// TwinCAT 3 PLC project PLC_ST01
// ProgramVersion: 3.1.4024.0
// libraries:
//   Base Objects Library, * (JABIL RAC LATAM)
//   Tc2_MC2, * (Beckhoff Automation GmbH)
//   Tc2_Standard, * (Beckhoff Automation GmbH)
//   Tc2_System, * (Beckhoff Automation GmbH)
//   Tc3_Module, * (Beckhoff Automation GmbH)
// project tree:
//   / PlcST01Task.TcTTO
//   POUs/00-MainPRG/ MAIN_ST01.TcPOU
//   POUs/01-FunctionBlocks/MaterialAssembly/ FB_ControllerAsm.TcPOU, FB_EndcapAsm.TcPOU
//   POUs/01-FunctionBlocks/MaterialSupply/ FB_BatterySupply.TcPOU, FB_ControllerSupply.TcPOU, FB_LoadStation.TcPOU
// real-time tasks:
//   TASK PlcST01Task: cycle T#10ms, priority 20, ADS port 350
//   TASK PlcST02Task: cycle T#10ms, priority 21, ADS port 351
//   TASK PlcST03Task: cycle T#10ms, priority 22, ADS port 352
// motion (NC):
//   TASK NC-Task 1 SAF: cycle T#2ms, priority 4, ADS port 501
//   TASK NC-Task 1 SVB: cycle T#10ms, priority 8, ADS port 511
//   AXIS Axis 1 (id 1)
//     OtherSettings: AllowMotionCmdToSlave=true
//     encoder EncType=19
//       EncPara: MaxCount=#xffffffff
//     drive DrvType=16
//       DrvPara: MaxCount=#xffffffff, DriveControlDWord=#x00000100
//         Analog: TorqueSetpointScale=10, ScaleFactorActTorque=0.1
//         TimeComp: TaskDelayCycles=1
//     controller CtrType=1
//       CtrPara: PriorControlFactor=1
//         Observer: BandWidth=20
//   AXIS Axis 2 (id 2)
//     OtherSettings: AllowMotionCmdToSlave=true
//     encoder EncType=19
//       EncPara: MaxCount=#xffffffff
//     drive DrvType=16
//       DrvPara: MaxCount=#xffffffff, DriveControlDWord=#x00000100
//         Analog: TorqueSetpointScale=10, ScaleFactorActTorque=0.1
//         TimeComp: TaskDelayCycles=1
//     controller CtrType=1
//       CtrPara: PriorControlFactor=1
//         Observer: BandWidth=20
//   AXIS Axis 3 (id 3)
//     OtherSettings: AllowMotionCmdToSlave=true
//     encoder EncType=19
//       EncPara: MaxCount=#xffffffff
//     drive DrvType=16
//       DrvPara: MaxCount=#xffffffff, DriveControlDWord=#x00000100
//         Analog: TorqueSetpointScale=10, ScaleFactorActTorque=0.1
//         TimeComp: TaskDelayCycles=1
//     controller CtrType=1
//       CtrPara: PriorControlFactor=1
//         Observer: BandWidth=20
// I/O:
//   DEVICE Device 1 (EtherCAT), AmsNetId 192.168.0.6.4.1
//     Term 1 (EK1100) [EK1100 EtherCAT Coupler (2A E-Bus)]
//       Term 2 (EL6910) [EL6910, TwinSAFE PLC]
//       Term 3 (EL1904) [EL1904, 4 Ch. Safety Input 24V, TwinSAFE]
//         modules: Module 1 (FSOES)
//       Term 4 (EL1904) [EL1904, 4 Ch. Safety Input 24V, TwinSAFE]
//         modules: Module 1 (FSOES)
//       Term 5 (EL1904) [EL1904, 4 Ch. Safety Input 24V, TwinSAFE]
//         modules: Module 1 (FSOES)
//       Term 6 (EL1904) [EL1904, 4 Ch. Safety Input 24V, TwinSAFE]
//         modules: Module 1 (FSOES)
//       Term 7 (EL1904) [EL1904, 4 Ch. Safety Input 24V, TwinSAFE]
//         modules: Module 1 (FSOES)
//       Term 8 (EL1904) [EL1904, 4 Ch. Safety Input 24V, TwinSAFE]
//         modules: Module 1 (FSOES)
//       Term 9 (EL1904) [EL1904, 4 Ch. Safety Input 24V, TwinSAFE]
//         modules: Module 1 (FSOES)
//       Term 10 (EL1904) [EL1904, 4 Ch. Safety Input 24V, TwinSAFE]
//         modules: Module 1 (FSOES)
//       Term 11 (EL9410) [EL9410 E-Bus Power Supplier  (Diagnostics)]
//       Term 12 (EL2904) [EL2904, 4 Ch. Safety Output 24V, 0.5A, TwinSAFE]
//         modules: Module 1 (FSOES), Module 2 (DO)
//       Term 13 (EL2904) [EL2904, 4 Ch. Safety Output 24V, 0.5A, TwinSAFE]
//         modules: Module 1 (FSOES), Module 2 (DO)
//       Term 14 (EL2904) [EL2904, 4 Ch. Safety Output 24V, 0.5A, TwinSAFE]
//         modules: Module 1 (FSOES), Module 2 (DO)
//       Term 15 (EL2904) [EL2904, 4 Ch. Safety Output 24V, 0.5A, TwinSAFE]
//         modules: Module 1 (FSOES), Module 2 (DO)
//       Term 16 (EL1809) [EL1809 16Ch. Dig. Input 24V, 3ms]
//       Term 17 (EL1809) [EL1809 16Ch. Dig. Input 24V, 3ms]
//       Term 18 (EL1809) [EL1809 16Ch. Dig. Input 24V, 3ms]
//       Term 19 (EL1809) [EL1809 16Ch. Dig. Input 24V, 3ms]
//       Term 20 (EL1809) [EL1809 16Ch. Dig. Input 24V, 3ms]
//       Term 21 (EL1809) [EL1809 16Ch. Dig. Input 24V, 3ms]
//       Term 22 (EL1809) [EL1809 16Ch. Dig. Input 24V, 3ms]
//       Term 23 (EL9410) [EL9410 E-Bus Power Supplier  (Diagnostics)]
//       Term 24 (EL1809) [EL1809 16Ch. Dig. Input 24V, 3ms]
//       Term 25 (EL1809) [EL1809 16Ch. Dig. Input 24V, 3ms]
//       Term 26 (EL1809) [EL1809 16Ch. Dig. Input 24V, 3ms]
//       Term 27 (EL2809) [EL2809 16Ch. Dig. Output 24V, 0.5A]
//       Term 28 (EL2809) [EL2809 16Ch. Dig. Output 24V, 0.5A]
//       Term 29 (EL2809) [EL2809 16Ch. Dig. Output 24V, 0.5A]
//       Term 30 (EL2809) [EL2809 16Ch. Dig. Output 24V, 0.5A]
//       Term 31 (EL2809) [EL2809 16Ch. Dig. Output 24V, 0.5A]
//       Term 32 (EL2809) [EL2809 16Ch. Dig. Output 24V, 0.5A]
//       Term 33 (EL2809) [EL2809 16Ch. Dig. Output 24V, 0.5A]
//       Term 34 (EL2809) [EL2809 16Ch. Dig. Output 24V, 0.5A]
//       Term 35 (EL3062) [EL3062 2Ch. Ana. Input 0-10V]
//       Term 36 (EL6652) [EL6652 EtherNet/IP Scanner (Master)]
//       Term 40 (EL9011) [EL9011 End Terminal]
//     Drive 37 (MDDLT55BF) [MDDLT55BF]
//     Drive 38 (MADLT05BF) [MADLT05BF]
//     Drive 39 (MADLT05BF) [MADLT05BF]
//   DEVICE Device 1 (ECAT EIP Scanner (EL6652)), AmsNetId 192.168.0.6.2.1
//     Robot01_Controller // <INFO> 192.168.0.21, ABB Adapter (ProdCode: 1, Rev: 2.50, Mac: 74:fe:48:88:fe:f3) </INFO> <EDS> C:\TwinCAT\3.1\Config\Io\EtherNetIP\enip.eds </EDS>
//     Robot02_Battery // <INFO> 192.168.0.22, ABB Adapter (ProdCode: 1, Rev: 2.50, Mac: 74:fe:48:87:d9:ae) </INFO> <EDS> C:\TwinCAT\3.1\Config\Io\EtherNetIP\enip.eds </EDS>
//     Robot03_1-2 // <INFO> 192.168.0.23, ABB Adapter (ProdCode: 1, Rev: 2.50, Mac: 74:fe:48:88:fe:f0) </INFO> <EDS> C:\TwinCAT\3.1\Config\Io\EtherNetIP\enip.eds </EDS>
//     Robot04_2-3 // <INFO> 192.168.0.24, ABB Adapter (ProdCode: 1, Rev: 2.50, Mac: 74:fe:48:88:0a:25) </INFO> <EDS> C:\TwinCAT\3.1\Config\Io\EtherNetIP\enip.eds </EDS>
//     NX1P2_ControllerTFPLC // <INFO> 192.168.0.10, NX1P2 (ProdCode: 1675, Rev: 2.09, Mac: 3c:f7:d1:1e:14:dc) </INFO> <EDS> C:\TwinCAT\3.1\Config\Io\EtherNetIP\ </EDS>
//     NX1P2_BatteryTrayFeederPLC // <INFO> 192.168.0.13, NX1P2 (ProdCode: 1675, Rev: 2.09, Mac: 3c:f7:d1:16:20:93) </INFO> <EDS> C:\TwinCAT\3.1\Config\Io\EtherNetIP\ </EDS>
// variable links:
//   NC-Task 1 SAF/Axes/Axis 1 <-> Device 1 (EtherCAT)/Drive 37 (MDDLT55BF)
//     Drive/Inputs/In/nDataIn1 <-> Transmit PDO mapping 1/Following error actual value
//     Drive/Inputs/In/nState1 <-> Transmit PDO mapping 1/Statusword
//     Drive/Inputs/In/nState2 <-> Transmit PDO mapping 1/Statusword @bit 8
//     Drive/Inputs/In/nState4 @bit 1 <-> WcState/InputToggle
//     Drive/Inputs/In/nState4 <-> WcState/WcState
//     Drive/Inputs/In/nState5 <-> Transmit PDO mapping 1/Modes of operation display
//     Drive/Outputs/Out/nCtrl1 <-> Receive PDO mapping 1/Controlword
//     Drive/Outputs/Out/nCtrl2 <-> Receive PDO mapping 1/Controlword @bit 8
//     Drive/Outputs/Out/nCtrl5 <-> Receive PDO mapping 1/Modes of operation
//     Drive/Outputs/Out/nDataOut1 <-> Receive PDO mapping 1/Target position
//     Enc/Inputs/In/nDataIn1 <-> Transmit PDO mapping 1/Position actual value
//     Enc/Inputs/In/nDataIn3 <-> Transmit PDO mapping 1/Touch probe pos1 pos value
//     Enc/Inputs/In/nState4 @bit 1 <-> WcState/InputToggle
//     Enc/Inputs/In/nState4 <-> WcState/WcState
//     Enc/Inputs/In/nState5 <-> Transmit PDO mapping 1/Touch probe status
//     Enc/Inputs/In/nState6 <-> Transmit PDO mapping 1/Touch probe status @bit 8
//     Enc/Outputs/Out/nCtrl5 <-> Receive PDO mapping 1/Touch probe function
//     Enc/Outputs/Out/nCtrl6 <-> Receive PDO mapping 1/Touch probe function @bit 8
//   NC-Task 1 SAF/Axes/Axis 2 <-> Device 1 (EtherCAT)/Drive 38 (MADLT05BF)
//     Drive/Inputs/In/nDataIn1 <-> Transmit PDO mapping 1/Following error actual value
//     Drive/Inputs/In/nState1 <-> Transmit PDO mapping 1/Statusword
//     Drive/Inputs/In/nState2 <-> Transmit PDO mapping 1/Statusword @bit 8
//     Drive/Inputs/In/nState4 @bit 1 <-> WcState/InputToggle
//     Drive/Inputs/In/nState4 <-> WcState/WcState
//     Drive/Inputs/In/nState5 <-> Transmit PDO mapping 1/Modes of operation display
//     Drive/Outputs/Out/nCtrl1 <-> Receive PDO mapping 1/Controlword
//     Drive/Outputs/Out/nCtrl2 <-> Receive PDO mapping 1/Controlword @bit 8
//     Drive/Outputs/Out/nCtrl5 <-> Receive PDO mapping 1/Modes of operation
//     Drive/Outputs/Out/nDataOut1 <-> Receive PDO mapping 1/Target position
//     Enc/Inputs/In/nDataIn1 <-> Transmit PDO mapping 1/Position actual value
//     Enc/Inputs/In/nDataIn3 <-> Transmit PDO mapping 1/Touch probe pos1 pos value
//     Enc/Inputs/In/nState4 @bit 1 <-> WcState/InputToggle
//     Enc/Inputs/In/nState4 <-> WcState/WcState
//     Enc/Inputs/In/nState5 <-> Transmit PDO mapping 1/Touch probe status
//     Enc/Inputs/In/nState6 <-> Transmit PDO mapping 1/Touch probe status @bit 8
//     Enc/Outputs/Out/nCtrl5 <-> Receive PDO mapping 1/Touch probe function
//     Enc/Outputs/Out/nCtrl6 <-> Receive PDO mapping 1/Touch probe function @bit 8
//   NC-Task 1 SAF/Axes/Axis 3 <-> Device 1 (EtherCAT)/Drive 39 (MADLT05BF)
//     Drive/Inputs/In/nDataIn1 <-> Transmit PDO mapping 1/Following error actual value
//     Drive/Inputs/In/nState1 <-> Transmit PDO mapping 1/Statusword
//     Drive/Inputs/In/nState2 <-> Transmit PDO mapping 1/Statusword @bit 8
//     Drive/Inputs/In/nState4 @bit 1 <-> WcState/InputToggle
//     Drive/Inputs/In/nState4 <-> WcState/WcState
//     Drive/Inputs/In/nState5 <-> Transmit PDO mapping 1/Modes of operation display
//     Drive/Outputs/Out/nCtrl1 <-> Receive PDO mapping 1/Controlword
//     Drive/Outputs/Out/nCtrl2 <-> Receive PDO mapping 1/Controlword @bit 8
//     Drive/Outputs/Out/nCtrl5 <-> Receive PDO mapping 1/Modes of operation
//     Drive/Outputs/Out/nDataOut1 <-> Receive PDO mapping 1/Target position
//     Enc/Inputs/In/nDataIn1 <-> Transmit PDO mapping 1/Position actual value
//     Enc/Inputs/In/nDataIn3 <-> Transmit PDO mapping 1/Touch probe pos1 pos value
//     Enc/Inputs/In/nState4 @bit 1 <-> WcState/InputToggle
//     Enc/Inputs/In/nState4 <-> WcState/WcState
//     Enc/Inputs/In/nState5 <-> Transmit PDO mapping 1/Touch probe status
//     Enc/Inputs/In/nState6 <-> Transmit PDO mapping 1/Touch probe status @bit 8
//     Enc/Outputs/Out/nCtrl5 <-> Receive PDO mapping 1/Touch probe function
//     Enc/Outputs/Out/nCtrl6 <-> Receive PDO mapping 1/Touch probe function @bit 8
//   PLC_ST01/PLC_ST01 Instance <-> Device 1 (ECAT EIP Scanner (EL6652))/Robot02_Battery
//     PlcST01Task Inputs/MAIN_ST01.fbBatterySupply.fbRobot.RobotIO.eipInputs <-> Connection 2 (Input/Output)/Inputs/inputRaw

CONFIGURATION PLC_ST01
    RESOURCE PLC ON TwinCAT3
        TASK PlcST01Task(INTERVAL := T#10ms, PRIORITY := 20);
        PROGRAM MAIN_ST01 WITH PlcST01Task : MAIN_ST01;
    END_RESOURCE
END_CONFIGURATION

// ---- POUs/00-MainPRG/MAIN_ST01.TcPOU
PROGRAM MAIN_ST01
VAR
	fbStation01							: RACBaseObjects.FB_Station;
	fbConveyor							: RACBaseObjects.FB_Conveyor;
	fbControllerSupply					: FB_ControllerSupply;
	fbBatterySupply						: FB_BatterySupply;
	fbEndcapAsm							: FB_EndcapAsm;
	fbControllerAsm						: FB_ControllerAsm;
	fbLoadStation						: FB_LoadStation;
	
	// Input from ST02
	ST02_initFinished					AT%I* : BOOL;
	ST02_mtrlReq						AT%I* : BOOL;
	
	// Estop declaration
	bEStopLoad							AT%I*	: BOOL;
	bEStopUserInterface					AT%I*	: BOOL;
	
	// Door no contact declaration
	
	// Interlock inputs declaration
	
END_VAR

	fbStation01(						bInitFinished:=fbControllerSupply.bInit_Finished AND fbBatterySupply.bInit_Finished AND fbConveyor.bInit_Finished,
										EmergencyStop:=bEStopLoad OR bEStopUserInterface,
										safetyReady:=TRUE,
										Interlock:=TRUE);

	fbConveyor(							sDeviceID:='',
										bStopExecution:=fbStation01.bStop,
										bAlarmReset:=fbStation01.bAlarmReset,
										diStationState:=fbStation01.diStationState,
										bInit_StartPermissive:=fbLoadStation.bInit_Finished AND fbEndcapAsm.bInit_Finished AND fbControllerAsm.bInit_Finished AND fbBatterySupply.bInit_Finished AND ST02_initFinished,
										bIn_SafeToMove:=FALSE,
										bIn_AllProcessComplete:=FALSE,
										lrDistance:=0,
										lrOffsetPos:=0,
										bIn_IsClamped:=FALSE,
										bIn_IsUnclamped:=FALSE);

	fbLoadStation(						sDeviceID:='',
										bStopExecution:=fbStation01.bStop,
										bAlarmReset:=fbStation01.bAlarmReset,
										diStationState:=fbStation01.diStationState,
										bInit_StartPermissive := TRUE,
										bDisableScan := TRUE,
										bIn_MovePermisive := FALSE,
										bIn_CvyStepDone := FALSE);

	fbEndcapAsm(						sDeviceID:='',
										bStopExecution:=fbStation01.bStop,
										bAlarmReset:=fbStation01.bAlarmReset,
										diStationState:=fbStation01.diStationState,
										bInit_StartPermissive:=TRUE,
										bSafetyBoxPlace_permissive :=TRUE);
	
										
	fbControllerSupply(					sDeviceID:='',
										bStopExecution:=fbStation01.bStop,
										bAlarmReset:=fbStation01.bAlarmReset,
										diStationState:=fbStation01.diStationState,
										bInit_StartPermissive:=TRUE,
										bSafetyBoxPlace_permissive:=FALSE,
										bPlace_MaterialRequest:=FALSE);
										
	fbControllerAsm(					sDeviceID:='',
										bStopExecution:=fbStation01.bStop,
										bAlarmReset:=fbStation01.bAlarmReset,
										diStationState:=fbStation01.diStationState,
										bInit_StartPermissive:=TRUE,
										sSerialReceived:=fbControllerSupply.sPieceSN,	
										bIn_RailReady:=fbConveyor.bOut_MoveDone);
										
	fbBatterySupply(					sDeviceID:='',
										bStopExecution:=fbStation01.bStop,
										bAlarmReset:=fbStation01.bAlarmReset,
										diStationState:=fbStation01.diStationState,
										bInit_StartPermissive:=TRUE,
										bSafetyBoxPlace_permissive := FALSE,
										bPlace_MaterialRequest := TRUE);

END_PROGRAM

// ---- POUs/01-FunctionBlocks/MaterialSupply/FB_ControllerSupply.TcPOU
FUNCTION_BLOCK FB_ControllerSupply EXTENDS RACBaseObjects.FB_Machine
VAR_INPUT
	bSafetyBoxPlace_Permissive			: BOOL;
	bPlace_MaterialRequest				: BOOL;
END_VAR
VAR_OUTPUT
	bSafetyBoxPlace_OutOfZone			: BOOL;
	sPieceSN							: STRING;
	bPlace_Done							: BOOL;
END_VAR
VAR
	fbTrayFeeder						: RACBaseObjects.FB_TrayFeeder;
	fbRobot								: RACBaseObjects.FB_Robot;
	fbScanner							: RACBaseObjects.FB_Scanner;
	
	// Reject on belt in tray feeder safery box permissive
	bSafetyBoxReject_permissive			AT%I*	: BOOL;
	// Reject on belt in tray feeder material request
	bReject_MaterialRequest				AT%I*	: BOOL;
	// Reject on belt in tray feeder out of safery box
	bSafetyBoxReject_OutOfZone			AT%Q*	: BOOL;
	// Reject on belt in tray feeder reject done
	bReject_Done						AT%Q*	: BOOL;
	
	// Auto procees is scanning
	bScann								: BOOL;
	
	// OK esponse from Acuram MES consultimng
	bPieceIsGood						: BOOL;
	// NG esponse from Acuram MES consultimng
	bPieceIsNG							: BOOL;
	
	// Auxiliar bool array for reject places inputs
	bAvailableNests						: ARRAY[0..7] OF BOOL;
END_VAR

SUPER^.MachineMain();
//	Tray Feeder instance
	fbTrayFeeder(						sDeviceID:=	'01',
										bStopExecution:=bStopExecution,
										bAlarmReset:=bAlarmReset,
										diStationState:=diStationState,
										bInit_StartPermissive:=fbRobot.bInit_Finished,
										bSafetyBoxDeliver_permissive:=fbRobot.bSafetyBoxPick_OutOfZone,
										bChangeTrayRequest:=fbRobot.bPick_AllMaterialPicked);

//	Robot instance
	fbRobot(							sDeviceID:=	'01',
										bStopExecution:=bStopExecution,
										bAlarmReset:=bAlarmReset,
										diStationState:=diStationState,
										bInit_StartPermissive:=bInit_StartPermissive,
										bSafetyBoxPick_Permissive:=fbTrayFeeder.bSafetyBoxDeliver_isSafe,
										bSafetyBoxPlace_Permissive:=bSafetyBoxPlace_permissive,
										bSafetyBoxReject_Permissive:=bSafetyBoxReject_Permissive,
										bOKMaterialReadyToPick:=fbTrayFeeder.bMaterial_ReadyToPick,
										bNGMaterialReadyToPick:=FALSE,
										bPiceIsGood:=bPieceIsGood,
										bPiceIsNG:=bPieceIsNG,
										bPlace_MaterialRequest:=bPlace_MaterialRequest,
										bReject_MaterialRequest:=bAvailableNests,
										bSafetyBoxPlace_OutOfZone=>bSafetyBoxPlace_OutOfZone,
										bSafetyBoxReject_OutOfZone=>bSafetyBoxReject_OutOfZone,
										bPlace_Done=>bPlace_Done,
										bReject_Done=>bReject_Done);

//	Scanner insance
	fbScanner(							sDeviceID:=	'03',
										bStopExecution:=bStopExecution,
										bAlarmReset:=bAlarmReset,
										bIn_Trigger:=bScann,
										bDisable:=FALSE,
										iTotalRetries:=2,
										Timeout:=t#1s);

METHOD Alarm
sAlarm:= CONCAT(STR1:=fbTrayFeeder.sAlarm, STR2:=fbRobot.sAlarm);
sAlarm:= CONCAT(STR1:=sAlarm,STR2:=fbScanner.sAlarm);
END_METHOD

METHOD Auto
//	When finish reading save the code in a var
	IF (fbRobot.diActualSeqStep=EN_RobotMessaging.waitingPieceStatus) THEN
		bScann:=TRUE;
		IF (fbScanner.bCompleted) AND (sPieceSN<>fbScanner.sCode) THEN
			sPieceSN:=fbScanner.sCode;
		END_IF
	END_IF

//	For clearing code in var
	IF (fbRobot.diActualSeqStep<>EN_RobotMessaging.waitingPieceStatus) AND (fbRobot.diActualSeqStep<>EN_RobotMessaging.placing) AND (fbRobot.diActualSeqStep<>EN_RobotMessaging.placeFinished) THEN
		bPieceIsGood:=FALSE;
		bPieceIsNG:=FALSE;
		sPieceSN:='';
	END_IF
END_METHOD

METHOD Init
bInit_Finished:=fbTrayFeeder.bInit_Finished AND fbRobot.bInit_Finished AND fbScanner.bConnected;
END_METHOD

METHOD IO
//	For robot available places inputs
	bAvailableNests[0]					:= bReject_MaterialRequest;
	bAvailableNests[1]					:= FALSE;
	bAvailableNests[2]					:= FALSE;
	bAvailableNests[3]					:= FALSE;
	bAvailableNests[4]					:= FALSE;
	bAvailableNests[5]					:= FALSE;
	bAvailableNests[6]					:= FALSE;
	bAvailableNests[7]					:= FALSE;
END_METHOD

{warning 'Add method implementation '}
METHOD Manual
END_METHOD

{warning 'Add method implementation '}
METHOD Pause
END_METHOD

{warning 'Add method implementation '}
METHOD Stop
END_METHOD

END_FUNCTION_BLOCK

// ---- POUs/01-FunctionBlocks/MaterialSupply/FB_BatterySupply.TcPOU
FUNCTION_BLOCK FB_BatterySupply EXTENDS RACBaseObjects.FB_Machine
VAR_INPUT
	bSafetyBoxPlace_permissive			: BOOL;
	
	bPlace_MaterialRequest				: BOOL;
END_VAR
VAR_OUTPUT
	bSafetyBoxPlace_OutOfZone			: BOOL;
	
	sPieceSN							: STRING;
	sPieceOnGantrySN					: STRING;
	sPieceOnSliderSN					: STRING;
	
	bPlace_Done							: BOOL;
END_VAR
VAR
	fbTrayFeeder						: RACBaseObjects.FB_TrayFeeder;
	fbRobot								: RACBaseObjects.FB_Robot;
	fbScanner							: RACBaseObjects.FB_Scanner;
	
	// Auto procees is scanning
	bScann								: BOOL;
	
	// Auxiliar bool array for reject places inputs
	bAvailableNests						: ARRAY[0..7] OF BOOL;
END_VAR

SUPER^.MachineMain();
//	Tray Feeder instance
	fbTrayFeeder(						sDeviceID:=	'',
										bStopExecution:=bStopExecution,
										bAlarmReset:=bAlarmReset,
										diStationState:=diStationState,
										bInit_StartPermissive:=fbRobot.bInit_Finished,
										bSafetyBoxDeliver_permissive:=fbRobot.bSafetyBoxPick_OutOfZone,
										bChangeTrayRequest:=fbRobot.bPick_AllMaterialPicked);

//	Robot instance
//	fbRobot(							sDeviceID:=	'',
//										bStopExecution:=bStopExecution,
//										bAlarmReset:=bAlarmReset,
//										diStationState:=diStationState,
//										bInit_StartPermissive:=bInit_StartPermissive,
//										bSafetyBoxPick_Permissive:=fbTrayFeeder.bSafetyBoxDeliver_isSafe,
//										bSafetyBoxPlace_Permissive:=bSafetyBoxPlace_permissive,
//										bSafetyBoxReject_Permissive:=FALSE,
//										bOKMaterialReadyToPick:=fbTrayFeeder.bMaterial_ReadyToPick,
//										bNGMaterialReadyToPick:=FALSE,
//										bPiceIsGood:=TRUE,
//										bPiceIsNG:=FALSE,
//										bPlace_MaterialRequest:=bPlace_MaterialRequest,
//										bReject_MaterialRequest:=bAvailableNests,
//										bSafetyBoxPlace_OutOfZone=>bSafetyBoxPlace_OutOfZone,
//										bPlace_Done=>bPlace_Done);

//	Scanner insance
	fbScanner(							sDeviceID:=	'',
										bStopExecution:=bStopExecution,
										bAlarmReset:=bAlarmReset,
										bIn_Trigger:=bScann,
										bDisable:=FALSE,
										iTotalRetries:=2,
										Timeout:=t#1s);

METHOD Alarm
sAlarm:= CONCAT(STR1:=fbTrayFeeder.sAlarm, STR2:=fbRobot.sAlarm);
sAlarm:= CONCAT(STR1:=sAlarm,STR2:=fbScanner.sAlarm);
END_METHOD

METHOD Auto
VAR
END_VAR
//	When slider is not taking piece, reaching delivery position or delivering unit, clear piece on slider code var
	IF (fbTrayFeeder.diActualSeqStep<>1110) AND (fbTrayFeeder.diActualSeqStep<>1120) AND (fbTrayFeeder.diActualSeqStep<>1130) THEN
		sPieceSN:='';
	END_IF

//	When finish reading save the code in a var
	IF fbTrayFeeder.diActualSeqStep=1110 THEN
		bScann:=TRUE;
		IF (fbScanner.bCompleted) AND (sPieceSN<>fbScanner.sCode) THEN
			sPieceSN:=fbScanner.sCode;
		END_IF
	END_IF

//	When gantry takes the battery translate last serial code readed
	IF (fbTrayFeeder.diActualSeqStep=1130) AND (sPieceOnGantrySN=sPieceSN) THEN
		sPieceOnGantrySN:=sPieceSN;
	END_IF

//	When gantry release the battery translate serial code to other var
	IF (fbTrayFeeder.diActualSeqStep=1150) AND (sPieceOnSliderSN<>sPieceOnGantrySN) THEN
		sPieceOnSliderSN:=sPieceOnGantrySN;
	END_IF
END_METHOD

METHOD Init
bInit_Finished:=fbTrayFeeder.bInit_Finished AND fbRobot.bInit_Finished AND fbScanner.bConnected;
END_METHOD

METHOD IO
//	For robot available places inputs
	bAvailableNests[0]					:= FALSE;
	bAvailableNests[1]					:= FALSE;
	bAvailableNests[2]					:= FALSE;
	bAvailableNests[3]					:= FALSE;
	bAvailableNests[4]					:= FALSE;
	bAvailableNests[5]					:= FALSE;
	bAvailableNests[6]					:= FALSE;
	bAvailableNests[7]					:= FALSE;
END_METHOD

{warning 'Add method implementation '}
METHOD Manual
END_METHOD

{warning 'Add method implementation '}
METHOD Pause
END_METHOD

{warning 'Add method implementation '}
METHOD Stop
END_METHOD

END_FUNCTION_BLOCK

// ---- POUs/01-FunctionBlocks/MaterialAssembly/FB_EndcapAsm.TcPOU
FUNCTION_BLOCK INTERNAL FB_EndcapAsm EXTENDS RACBaseObjects.FB_Machine
VAR_INPUT
	bSafetyBoxPlace_permissive			: BOOL;
END_VAR
VAR_OUTPUT
	bOutEndcapAsm_Done 					: BOOL;
END_VAR
VAR
	bIsEndcapInFeedPosition		AT %I*		: BOOL;
	bIsEndcapInAssemblyPos		AT %I*		: BOOL;
	bFirstPositionSensor 		AT %I*		: BOOL;		
				
	//Is rail in position and clamped
	bRailReadyToAssembly					: BOOL;
	//Assembly side is ready to receive
	bAsmReadyToReceive						: BOOL;
	//Feed side with endcap ready
	bFeedReadyToSend						: BOOL;
	//The endcap is assembled on the rail
	bEndcapInRailDone						: BOOL;
	
	//Local process control
	bRemoveBottomSupport					: BOOL;
	bEndcapAssembled						: BOOL;
	bIsClampedOk							: BOOL;
	bIsReleased								: BOOL;
	bIsBottomClampRelease					: BOOL;								
	bEndcapPasses							: BOOL;		
	
	//Control steps for sub routines
	iStepAsm								: USINT;
	iStepFeed								: USINT;
	iStepRail								: USINT;
	
	//Timer to confirm endcap in position
	tmrPosition								: TON;
	tmrBowl									: TP;
	time_EC_DelayPosition					: TIME		:= T#500MS;
		
	//Devices
	
	//Bowl control structure, validate signals and control system1		
	bowlControl								: ST_BowlFeeder;	
	//Rail side for clamp support top cylinder
	Cyl_ClampRail_Top						: FB_Cylinder;
	//Rail side for clamp support bottom cylinder
	Cyl_ClampRail_Bot						: FB_Cylinder;		
	//Send endcap from bowl rail to assembly align
	Cyl_FeedEndcap							: FB_Cylinder;	
	//Push endcap for assembly with the rail 
	Cyl_PushEndcap							: FB_Cylinder;	
	//Endcap feeding guide during alignment process
	Cyl_SupportEndcap_Top					: FB_Cylinder;
	//Bottom alignment guide and pin button release 
	Cyl_SupportEndcap_Bot					: FB_Cylinder;

	bOut_ProcessComplete					: BOOL;
	bOut_ProcessOnFail						: BOOL;
	bOut_ReadyToReceive						: BOOL;
	bIn_UnitReady							: BOOL;
	bIn_UnitOnFail							: BOOL;
	
	//Manual operations
	bIn_Manual_ClampRail				: BOOL;
	bIn_Manual_UnclampRail				: BOOL;	
	bIn_ManualRun						: BOOL;		
	
	
END_VAR

SUPER^.MachineMain();

//Run FB and assign safety permisives


Cyl_ClampRail_Top();

Cyl_ClampRail_Bot();

//Set the permisive output directly from the cylinder sensors
bSafetyBoxPlace_Permissive := (Cyl_ClampRail_Top.bIsRetracted AND
							Cyl_ClampRail_Bot.bIsRetracted AND
							Cyl_PushEndcap.bIsRetracted);

METHOD Alarm
END_METHOD

METHOD Auto

VAR
	Seq_Endcap: INT;
END_VAR
//Call sub process
THIS^.Seq_EndcapFeed(bIsManual := TRUE);			//Feed endcap from bowl to assembly process
THIS^.Seq_EndcapAsm(bIsManual := TRUE);			//Endcap assembly process
THIS^.Seq_Auto_Rail();			//Clamp rail
THIS^.Seq_Auto_BowlFeeder();	//Bowl feeder control
END_METHOD

METHOD ClampRail : BOOL
//Top and bottom clamp
Cyl_ClampRail_Top.bExtendRequest:= TRUE;
Cyl_ClampRail_Bot.bExtendRequest:= TRUE;

ClampRail:=  Cyl_ClampRail_Top.bIsExtended AND Cyl_ClampRail_Bot.bIsExtended;
END_METHOD

METHOD fn_CancelCylinderMoves
VAR
	r_trig					: R_TRIG;
END_VAR
r_trig(CLK:= TRUE);
//Stop moves only once
IF r_trig.Q THEN
				
	Cyl_ClampRail_Bot.bExtendRequest:= FALSE;
	Cyl_ClampRail_Bot.bRetractRequest:= FALSE;
	
	Cyl_ClampRail_Top.bExtendRequest:= FALSE;
	Cyl_ClampRail_Top.bRetractRequest:= FALSE;
	
	Cyl_FeedEndcap.bExtendRequest:= FALSE;
	Cyl_FeedEndcap.bRetractRequest:= FALSE;
	
	Cyl_PushEndcap.bExtendRequest:= FALSE;
	Cyl_PushEndcap.bRetractRequest:= FALSE;
	
	Cyl_SupportEndcap_Bot.bExtendRequest:= FALSE;
	Cyl_SupportEndcap_Bot.bRetractRequest:= FALSE;
	
	Cyl_SupportEndcap_Top.bExtendRequest:= FALSE;
	Cyl_SupportEndcap_Top.bRetractRequest:= FALSE;
END_IF
END_METHOD

 METHOD Init 

//VAR_OUTPUT
//	bOutReadyToRobotPlace: BOOL;
//END_VAR
CASE diActualSeqStep OF
	//Initial
		
	0:						//Reset variables		
		bInit_Finished := FALSE;
	     bOutEndcapAsm_Done:= FALSE;		
		diActualSeqStep:= 10;	
		
	10:						//Retract rail support				
		//Retract controller guide support
		Cyl_SupportEndcap_Top.bRetractRequest := TRUE;
		Cyl_SupportEndcap_Bot.bRetractRequest := TRUE;
							
		IF THIS^.UnclampRail() AND Cyl_SupportEndcap_Top.bIsRetracted AND Cyl_SupportEndcap_Bot.bIsRetracted THEN
			diActualSeqStep := 20;			
		END_IF
	
	20:						//Retract feed endcap cyl.		
		Cyl_FeedEndcap.bRetractRequest := TRUE;
		IF Cyl_FeedEndcap.bIsRetracted THEN 
			diActualSeqStep := 30;
		END_IF
		
	30:						//Retract push endcap to rail			
		Cyl_PushEndcap.bRetractRequest:= TRUE;
		IF Cyl_PushEndcap.bIsRetracted THEN
			diActualSeqStep:= 40;
		END_IF

	40:						//Initial done				 
		bInit_Finished:= TRUE;
		RETURN;
		
END_CASE
END_METHOD

METHOD IO
END_METHOD

METHOD Manual

VAR
	r_trigReset					: R_TRIG;
END_VAR

IF bIn_ManualRun THEN
	//Reset just once
	r_trigReset(CLK:= TRUE);
	IF r_trigReset.Q THEN
		iStepAsm:= 0;
		iStepFeed:= 0;				
	END_IF
	
	//Run sequences
	THIS^.Seq_EndcapAsm(bIsManual:= TRUE);		
	THIS^.Seq_EndcapAsm(bIsManual:= TRUE);		
END_IF


//Clamp rail
 IF bIn_Manual_ClampRail THEN
	 IF THIS^.ClampRail() THEN
		 bIn_Manual_ClampRail:= FALSE;
	 END_IF
 END_IF
 
 //Unclamp rail
 IF bIn_Manual_UnclampRail THEN
	 IF THIS^.UnclampRail() THEN
		 bIn_Manual_UnclampRail:= FALSE;
	 END_IF
 END_IF
END_METHOD

METHOD Pause
fn_CancelCylinderMoves();
END_METHOD

ACTION Seq_Auto_BowlFeeder:

//Bowl control
tmrbowl(PT:= T#500MS);
IF NOT bIsEndcapInFeedPosition OR tmrBowl.Q THEN
	bowlControl.bOut_Vibrate := TRUE;
	tmrBowl.IN:= TRUE;	
ELSE	
	tmrBowl.IN:= FALSE;
	bowlControl.bOut_Vibrate:= FALSE;
END_IF

//Alarm
IF bowlControl.bIn_NoMaterial THEN
	sAlarm:= 'Bowl feeder no material, please recharge';
	
ELSIF bowlControl.bIn_LowLevelMaterial THEN 
	sAlarm:='Bowl feeder low level material';
		
ELSE 
	sAlarm:= '';
END_IF
END_ACTION

ACTION Seq_Auto_Rail:
CASE iStepRail OF
	
	0:						//Reset variables				
		bOut_ProcessComplete:= FALSE;
		bOut_ProcessOnFail:= FALSE;
		bOut_ReadyToReceive:= FALSE;
		bRailReadyToAssembly:= FALSE;	
		iStepRail:= 10;
				
	10:						//Check status			
		iStepRail:= 20;
		
	20: 					//Retract clamps of rail
		IF THIS^.UnclampRail() THEN
			iStepRail := 30;
		END_IF	
		
	30:						//Wait for new rail and ok to process			
//		IF bIn_RailReady THEN
			IF RACBaseObjects.GVL_Rails.Nests[RACBaseObjects.Constants.EndcapAsmPos].okToProcess AND NOT bIn_UnitOnFail THEN
				iStepRail:= 40;			
			ELSIF bIn_UnitOnFail OR NOT RACBaseObjects.GVL_Rails.Nests[RACBaseObjects.Constants.EndcapAsmPos].okToProcess  THEN				
				iStepRail:= 60;				
			END_IF			 
//		END_IF
		
	40:						//Clamp rail		
		IF THIS^.ClampRail() THEN			
			iStepRail := 50;
		END_IF	
		
	50:						//Ready to controller assembly
		bRailReadyToAssembly:= TRUE;
		IF bEndcapInRailDone THEN
			bRailReadyToAssembly:= FALSE;
			iStepRail:= 60;
		END_IF
		
 	60: 					//Retract clamps
		IF THIS^.UnclampRail() THEN
			iStepRail:= 70;
		END_IF
		
	70:						//Send rail assembly done and wait until not rail in position
	   	bOut_ProcessComplete := TRUE;
		
		IF NOT bIn_UnitReady AND NOT bIn_UnitOnFail THEN
			bOut_ProcessComplete := FALSE;
			iStepRail:=80;
		END_IF

	80:						//Return to start
		iStepRail:= 0;
		
END_CASE
END_ACTION

METHOD PRIVATE Seq_EndcapAsm : BOOL
VAR_INPUT
	bIsManual			:BOOL 		:= FALSE;
END_VAR
CASE iStepAsm OF

	0:						//Reset variables
		bOut_ProcessComplete:= FALSE;
		bOut_ProcessOnFail:= FALSE;
		bOut_ReadyToReceive:= FALSE;
		bAsmReadyToReceive:= FALSE;
		
		iStepAsm:= 10;

	10:						//Check status
		iStepAsm:=20;
		
	20:						//Retract push cylinder
		Cyl_PushEndcap.bRetractRequest := TRUE;
		IF Cyl_PushEndcap.bIsRetracted THEN
			iStepAsm:= 30;
		END_IF

	30:						//Extend Endcap guides
		Cyl_SupportEndcap_Top.bExtendRequest := TRUE;
		Cyl_SupportEndcap_Bot.bExtendRequest := TRUE;
		
		IF Cyl_SupportEndcap_Top.bIsExtended AND Cyl_SupportEndcap_Bot.bIsExtended THEN
			iStepAsm:= 40;
		END_IF

	40:						//Send ready to receive and wait for endcap
		bAsmReadyToReceive:= TRUE;
		IF bIsEndcapInAssemblyPos THEN
			bAsmReadyToReceive:= FALSE;
			iStepAsm:= 50;
		END_IF
		
	50:						//Confirm feed side doesn't be ready
		IF NOT bFeedReadyToSend THEN
			iStepAsm:= 60;
		END_IF

	60:						//Wait for rail ready to assembly
		IF bRailReadyToAssembly THEN
			iStepAsm:= 70;
		END_IF
		
	70:						//Retract bottom support
		Cyl_SupportEndcap_Bot.bRetractRequest:= TRUE;
		IF Cyl_SupportEndcap_Bot.bIsRetracted THEN
			Cyl_SupportEndcap_Bot.bRetractRequest:= FALSE;
			iStepAsm:= 80;
		END_IF
		
	80:						//Push endcap into the rail
		Cyl_PushEndcap.bExtendRequest:= TRUE;
		IF Cyl_PushEndcap.bIsExtended THEN
			iStepAsm:= 90;
		END_IF
		
	90:						//Retract top guide
		Cyl_SupportEndcap_Top.bRetractRequest:= TRUE;
		IF Cyl_SupportEndcap_Top.bIsRetracted THEN			
			iStepAsm:= 100;
		END_IF
	
	100:						//Retract push
		Cyl_PushEndcap.bRetractRequest:= TRUE;
		IF Cyl_PushEndcap.bIsRetracted THEN
			iStepAsm:= 110;
		END_IF
	
	110:						//Send the assembly done
		bEndcapInRailDone:= TRUE;
		IF NOT bRailReadyToAssembly THEN
			iStepAsm:= 120;		
		END_IF
	
	120:						//Return to start
		iStepAsm:= 0;
		
END_CASE
END_METHOD

METHOD PRIVATE Seq_EndcapFeed : BOOL
VAR_INPUT
	bIsManual				:BOOL 		:= FALSE;	
END_VAR

VAR
	
END_VAR
CASE iStepFeed OF

	0:						//Reset variables		
		iStepFeed:= 10;

	10:						//Check status
		iStepFeed:= 20;
		
	20:						//Retract feed cylinder
		Cyl_FeedEndcap.bRetractRequest:= TRUE;
		IF Cyl_FeedEndcap.bIsRetracted THEN			
			iStepFeed:= 30;
		END_IF
	
	30:						//Wait for endcap in position
		IF bIsEndcapInFeedPosition THEN
			iStepFeed:= 40;
		END_IF

	40:						//Check Assembly position is ready to receive
		bFeedReadyToSend := TRUE;
		IF bAsmReadyToReceive THEN
			iStepFeed:= 50;
		END_IF
		
	50:						//Extend Endcap feed cylinder
		Cyl_FeedEndcap.bExtendRequest:= TRUE;
		IF Cyl_FeedEndcap.bIsExtended THEN
			Cyl_FeedEndcap.bExtendRequest:= FALSE;
			iStepFeed:= 60;
		END_IF		

	60:						//Confirm endcap in the next position
		IF NOT bAsmReadyToReceive THEN		
			iStepFeed:= 70;
		END_IF
		
	70:						//Retract feed cylinder
		Cyl_FeedEndcap.bRetractRequest:= TRUE;
		IF Cyl_FeedEndcap.bIsRetracted THEN
			bFeedReadyToSend:= FALSE;			
			iStepFeed:= 80;
		END_IF
			
	80:						//Return to start
		iStepFeed:= 0;


END_CASE
END_METHOD

METHOD Stop
fn_CancelCylinderMoves();
END_METHOD

METHOD UnclampRail : BOOL
		
//Top and bottom unclamp
Cyl_ClampRail_Top.bRetractRequest:= TRUE;
Cyl_ClampRail_Bot.bRetractRequest:= TRUE;

UnclampRail:= Cyl_ClampRail_Top.bIsRetracted AND Cyl_ClampRail_Bot.bIsRetracted;
END_METHOD

END_FUNCTION_BLOCK

// ---- POUs/01-FunctionBlocks/MaterialAssembly/FB_ControllerAsm.TcPOU
FUNCTION_BLOCK INTERNAL FB_ControllerAsm EXTENDS RACBaseObjects.FB_Machine

VAR_INPUT
	sSerialReceived						: STRING;	
	bIn_RailReady						: BOOL;
END_VAR

VAR_OUTPUT					
	bOut_ControlAsm_Done				: BOOL;
	bOut_ReadyToRobotPlace				: BOOL;
	bOut_RobotPermisive					: BOOL;
	bOutReadyToRobotPlace				: BOOL;
	bSafetyBoxPlace_OutOfZone 			: BOOL;

END_VAR

VAR		
	
	sSerialCenter						: STRING;
	sSerialAsm							: STRING;
	
	bInSensorBeforeFlipPos		AT %I*	: BOOL;
	bInSensorAfterFlipPos		AT %I*	: BOOL;
	bInSensorAlignedPos		 	AT %I*	: BOOL;
	bInMiddlePositionSensor 	AT %I*	: BOOL;	

	bRemoveBottomSupport				: BOOL;		
	bControllerInRailDone				: BOOL;	
	
	//Hanshake between subsequences							
	bReceiverReadyToSend				: BOOL;
	bCenterReadyToReceive				: BOOL;
	bCenterReadyToSend					: BOOL;
	bAsmReadyToReceive					: BOOL;	
	
	bRailReadyToAssembly				: BOOL;
	
	//Rail side vars	
	bIsClampedOk						: BOOL;
	bIsReleased							: BOOL;
	bIsBottomClampRelease				: BOOL;
	
	//Control steps 
	iStepAsm							: USINT;
	iStepCenter							: USINT;	
	iStepReceive						: USINT;
	iStepRail							: USINT;	
	
	//Remove noise timers
	tmrFlip								: TON;	
	tmrAsm								: TON;
	tmrCenter							: TON;
	
	tControlDelayPosition				: TIME		:= T#500MS;		
				
	//Devices	
	
	//Rail side for clamp support top cylinder
	Cyl_ClampRail_Top					: FB_Cylinder;
	//Rail side for clamp support bottom cylinder
	Cyl_ClampRail_Bot					: FB_Cylinder;
	//Rail side Busbar align support
	Cyl_BusbarSupport					: FB_Cylinder;	
	//Send controller from nest to assembly align
	Cyl_FeedControl						: FB_Cylinder;	
	//Push controller for assembly to the rail 
	Cyl_PushControl						: FB_Cylinder;
	//Flipper from robot place to nest
	Cyl_Flipper							: FB_Cylinder;
	//Controller guide during feed alignment process
	Cyl_SupportControl_Top				: FB_Cylinder;
	//Bottom alignment guide and pin button release 
	Cyl_SupportControl_Bot				: FB_Cylinder;				
	//Centering controller after flip
	Cyl_Center: FB_Cylinder;
	//Vacuum control
	Vacuum								: FB_Vacuum;
	
	//Manual operations
	bIn_Manual_ClampRail				: BOOL;
	bIn_Manual_UnclampRail				: BOOL;	
	bIn_ManualRun						: BOOL;		
					
END_VAR

//Run the main controller 
SUPER^.MachineMain();

//Run devices with their safety conditions
Cyl_ClampRail_Top(bPermisiveExtend:= Cyl_BusbarSupport.bIsRetracted);
Cyl_ClampRail_Bot(bPermisiveExtend:= Cyl_BusbarSupport.bIsRetracted);
Cyl_BusbarSupport(bPermisiveExtend:= Cyl_ClampRail_Top.bIsExtended AND Cyl_ClampRail_Bot.bIsExtended);

Cyl_SupportControl_Top(bPermisiveExtend:= Cyl_PushControl.bIsRetracted AND Cyl_FeedControl.bIsRetracted);
Cyl_SupportControl_Bot(bPermisiveExtend:= Cyl_PushControl.bIsRetracted AND Cyl_FeedControl.bIsRetracted);
Cyl_Center(bPermisiveExtend:= Cyl_Flipper.bIsRetracted and Cyl_FeedControl.bIsRetracted);

Cyl_Flipper(bPermisiveExtend:= Cyl_Center.bIsRetracted);
Cyl_PushControl(bPermisiveExtend:= Cyl_BusbarSupport.bIsExtended AND Cyl_FeedControl.bIsRetracted,
				bPermisiveRetract:= Cyl_FeedControl.bIsRetracted);
Cyl_FeedControl(bPermisiveExtend:= Cyl_PushControl.bIsRetracted AND Cyl_Center.bIsRetracted AND Cyl_Flipper.bIsRetracted,
				bPermisiveRetract:= Cyl_Center.bIsRetracted AND Cyl_Flipper.bIsRetracted);
				
//Vacuum();
Vacuum(	bStopExecution:=bStopExecution, 
		bAlarmReset:=bAlarmReset,
		Timeout:=T#1S);
		
//Robot permisive
bOut_RobotPermisive:= Cyl_Flipper.bIsRetracted;

//Conveyor permisive
bSafetyBoxPlace_OutOfZone:= Cyl_ClampRail_Top.bIsRetracted AND Cyl_ClampRail_Bot.bIsRetracted
						AND Cyl_BusbarSupport.bIsRetracted AND Cyl_PushControl.bIsRetracted;

METHOD Alarm
END_METHOD

METHOD Auto
//Call sub process
THIS^.Seq_CtrlReceive(bIsManual := FALSE);		//Receive from robot and flip controller
THIS^.Seq_CtrlCenter(bIsManual := FALSE);			//Receive from flipper, align and feed to assembly side
THIS^.Seq_CtrlAsm(bIsManual := FALSE);			//Guide controller and assembly on the rail
THIS^.Seq_Auto_Rail();			//Rail clamping
END_METHOD

METHOD ClampRail : BOOL
VAR_INPUT
END_VAR
//Top and bottom clamp
Cyl_ClampRail_Top.bExtendRequest := TRUE;
Cyl_ClampRail_Bot.bExtendRequest := TRUE;

IF Cyl_ClampRail_Top.bIsExtended AND Cyl_ClampRail_Bot.bIsExtended THEN
	//Extend busbar support
	Cyl_BusbarSupport.bExtendRequest:= TRUE;
	IF Cyl_BusbarSupport.bIsExtended THEN
		ClampRail:= TRUE;		
		RETURN;			
	END_IF
END_IF	
		
ClampRail:= FALSE;
END_METHOD

METHOD fn_CancelCylinderMoves
VAR
	r_trig					: R_TRIG;
END_VAR
r_trig(CLK:= TRUE);
//Stop moves only once
IF r_trig.Q THEN
	Cyl_BusbarSupport.bExtendRequest:= FALSE;
	Cyl_BusbarSupport.bRetractRequest:= FALSE;
	
	Cyl_Center.bRetractRequest:= FALSE;
	Cyl_Center.bExtendRequest:= FALSE;
	
	Cyl_ClampRail_Bot.bExtendRequest:= FALSE;
	Cyl_ClampRail_Bot.bRetractRequest:= FALSE;
	
	Cyl_ClampRail_Top.bExtendRequest:= FALSE;
	Cyl_ClampRail_Top.bRetractRequest:= FALSE;
	
	Cyl_FeedControl.bExtendRequest:= FALSE;
	Cyl_FeedControl.bRetractRequest:= FALSE;
	
	Cyl_Flipper.bExtendRequest:= FALSE;
	Cyl_Flipper.bRetractRequest:= FALSE;
	
	Cyl_PushControl.bExtendRequest:= FALSE;
	Cyl_PushControl.bRetractRequest:= FALSE;
	
	Cyl_SupportControl_Bot.bExtendRequest:= FALSE;
	Cyl_SupportControl_Bot.bRetractRequest:= FALSE;
	
	Cyl_SupportControl_Top.bExtendRequest:= FALSE;
	Cyl_SupportControl_Top.bRetractRequest:= FALSE;
END_IF
END_METHOD

METHOD Init

VAR
	bOutControlAsm_Done: BOOL;
END_VAR
CASE diActualSeqStep OF
	//Initial
	
	0:		//Reset variables
		bInit_Finished := FALSE;
		bOutControlAsm_Done	:= FALSE;
		bOut_ReadyToRobotPlace  := FALSE;		
		diActualSeqStep:= 10;	
	
	10:		//Retract bus bar support
		Cyl_BusbarSupport.bRetractRequest := TRUE;
		IF Cyl_BusbarSupport.bIsRetracted THEN			
			diActualSeqStep := 20;
		END_IF
	
	20:		//Retract rail support
		Cyl_ClampRail_Top.bRetractRequest:= TRUE;
		Cyl_ClampRail_Bot.bRetractRequest := TRUE;
	
			//Retract controller guide support
		Cyl_SupportControl_Top.bRetractRequest:= TRUE;
		Cyl_SupportControl_Bot.bRetractRequest:= TRUE;
		
			//Retract centering controller
		Cyl_Center.bRetractRequest:= TRUE;
		
		IF Cyl_ClampRail_Top.bIsRetracted AND Cyl_ClampRail_Bot.bIsRetracted
			AND Cyl_SupportControl_Top.bIsRetracted AND Cyl_SupportControl_Bot.bIsRetracted
			AND Cyl_Center.bIsRetracted THEN
			
			diActualSeqStep := 30;			
		END_IF
	
	30:		//Retract feed controller cyl.
		Cyl_FeedControl.bRetractRequest:= TRUE;
		IF Cyl_FeedControl.bIsRetracted THEN 			
			diActualSeqStep := 40;
		END_IF
		
	40:		//Retract push controller to rail
	
		Cyl_PushControl.bRetractRequest:= TRUE;
		IF Cyl_PushControl.bIsRetracted THEN			
			diActualSeqStep:= 50;
		END_IF
	
	50:		//Retract flipper
	
		Cyl_Flipper.bRetractRequest:= TRUE;
		IF Cyl_Flipper.bIsRetracted THEN			
			//Turn off vacuum valve without blow
			Vacuum.bGrip := FALSE;
			diActualSeqStep:= 60;
		END_IF
	
	60:		//Initial Done 
		bInit_Finished:= TRUE;
		diActualSeqStep:= 100;
		RETURN;
		
END_CASE
END_METHOD

METHOD IO
END_METHOD

METHOD Manual

VAR 
	r_trigReset							: R_TRIG;
END_VAR

IF bIn_ManualRun THEN
	//Reset just once
	r_trigReset(CLK:= TRUE);
	IF r_trigReset.Q THEN
		iStepAsm:= 0;
		iStepCenter:= 0;		
		iStepReceive:= 0;
	END_IF
	
	//Run sequences
	THIS^.Seq_CtrlReceive(bIsManual:= TRUE);	
	THIS^.Seq_CtrlCenter(bIsManual:= TRUE);		
	THIS^.Seq_CtrlAsm(bIsManual:= TRUE);		
END_IF


//Clamp rail
 IF bIn_Manual_ClampRail THEN
	 IF THIS^.ClampRail() THEN
		 bIn_Manual_ClampRail:= FALSE;
	 END_IF
 END_IF
 
 //Unclamp rail
 IF bIn_Manual_UnclampRail THEN
	 IF THIS^.UnclampRail() THEN
		 bIn_Manual_UnclampRail:= FALSE;
	 END_IF
 END_IF
END_METHOD

METHOD Pause
fn_CancelCylinderMoves();
END_METHOD

ACTION Seq_Auto_Rail:
CASE iStepRail OF
	
	0:						//Reset variables
		bOut_ControlAsm_Done:= FALSE;
		bRailReadyToAssembly:= FALSE;	
		iStepRail:= 10;
				
	10:						//Check status			
		iStepRail:= 20;
	
	20:						//Retract busbar support
		Cyl_BusbarSupport.bRetractRequest:= TRUE;
		IF Cyl_BusbarSupport.bIsRetracted THEN
			iStepRail:= 30;
		END_IF
	
	30:						//Retract rail clamps 
		Cyl_ClampRail_Top.bRetractRequest:= TRUE;
		Cyl_ClampRail_Bot.bRetractRequest:= TRUE;

		IF Cyl_ClampRail_Top.bIsRetracted AND Cyl_ClampRail_Bot.bIsRetracted THEN
			iStepRail := 40;
		END_IF	
		
	40:						//Wait for new rail in position and ok to process
		IF   bIn_RailReady AND  GVL_Rails.Nests[Constants.ControllerAsmPos].okToProcess THEN
			iStepRail:= 50;
		END_IF
		
	50:						//Clamp rail	
		IF 	THIS^.ClampRail() THEN
			
			iStepRail := 60;
		END_IF

//Ready to controller assembly
	60:
		bRailReadyToAssembly:= TRUE;
		IF bControllerInRailDone THEN
			bRailReadyToAssembly:= FALSE;
			iStepRail:= 70;
		END_IF
		
//Retract busbar
	70:
		IF THIS^.UnclampRail() THEN
			iStepRail:= 80;
		END_IF
 
//Send rail assembly done and wait until not rail in position
	80:
		  bOut_ControlAsm_Done:= TRUE;
		
		IF NOT bIn_RailReady THEN
			bOut_ControlAsm_Done:= FALSE;
			iStepRail:= 90;
		END_IF

//Return to start
	90:
		iStepRail:= 0;
		
END_CASE
END_ACTION

METHOD PRIVATE Seq_CtrlAsm
VAR_INPUT
	bIsManual				: BOOL			:= FALSE;
END_VAR
CASE iStepAsm OF

	0:							//Reset variables		
		bAsmReadyToReceive:= FALSE;			
		bControllerInRailDone:= FALSE;
		tmrAsm.IN:= FALSE;
		iStepAsm:= 10;
				
	10:							//Check status
		IF bInSensorAlignedPos THEN	//Controller in rail aligned pos
			//Avoid noise with the timer
			tmrAsm(IN:= TRUE, pt:= T#200MS);
			
			IF tmrAsm.Q THEN
				iStepAsm:= 40;
			END_IF				
					
		ELSE	//Nothing detected
			tmrAsm.IN:= FALSE;		
			iStepAsm:= 20;
		END_IF

	20:							//Confirm push cylinder retracted
		Cyl_PushControl.bRetractRequest:= TRUE;
		IF Cyl_PushControl.bIsRetracted THEN
			Cyl_PushControl.bRetractRequest:=FALSE;
			iStepAsm:= 30;
		END_IF
		
	30:							//Extend controller guide cylinders
		Cyl_SupportControl_Top.bExtendRequest:= TRUE;
		Cyl_SupportControl_Bot.bExtendRequest:= TRUE;
				
		IF Cyl_SupportControl_Top.bIsExtended AND Cyl_SupportControl_Bot.bIsExtended THEN						
			iStepAsm:= 40;									
		END_IF

	40:							//Wait for controller in position
		bAsmReadyToReceive:= TRUE;
		IF bInSensorAlignedPos AND NOT bCenterReadyToSend THEN			
			bAsmReadyToReceive:= FALSE;
			iStepAsm:= 50;			
		END_IF
		 
	50:							//Retract controller bottom support cylinder
		Cyl_SupportControl_Bot.bRetractRequest:= TRUE;
			IF Cyl_SupportControl_Bot.bIsRetracted THEN			
			 	iStepAsm:= 60;
		 	END_IF

	60:							//Wait for rail ready to assembly and clamped
		IF bRailReadyToAssembly OR bIn_ManualRun THEN
			istepAsm:= 70;
		END_IF
		
	70: 						//Push controller to the rail
		Cyl_PushControl.bExtendRequest:= TRUE;
		IF Cyl_PushControl.bIsExtended THEN
			Cyl_PushControl.bExtendRequest:= FALSE;
			istepAsm:= 80;
		END_IF
		
	80:							//If not in manual, update the serial on the gvl rail list 
		IF NOT bIn_ManualRun THEN
			GVL_Rails.Nests[Constants.ControllerAsmPos].controllerSerial:= sSerialAsm;
		END_IF
		iStepAsm:= 90;		
		
	90:							//Remove top controller guide and bottom rail support
		Cyl_SupportControl_Top.bRetractRequest:= TRUE;
		Cyl_ClampRail_Bot.bRetractRequest:= TRUE;
		tmrAsm(IN:= FALSE);
		
		IF Cyl_SupportControl_Top.bIsRetracted AND Cyl_ClampRail_Bot.bIsRetracted THEN			
			iStepAsm:= 100;			
		END_IF
		
	100:							//Confirm full controller assembly
		Cyl_PushControl.bExtendRequest:= TRUE;
		IF Cyl_PushControl.bIsExtended THEN
			
			tmrAsm(IN:= TRUE, pt:= T#100MS);
			IF tmrAsm.Q THEN				
				istepAsm:= 110;
			END_IF			
		END_IF

	110:							//Retract assembly side cylinders
		Cyl_PushControl.bRetractRequest:= TRUE;
		Cyl_SupportControl_Top.bRetractRequest:= TRUE;
		Cyl_SupportControl_Bot.bRetractRequest:= TRUE;
		
		IF Cyl_PushControl.bIsRetracted AND Cyl_SupportControl_Top.bIsRetracted AND Cyl_SupportControl_Bot.bIsRetracted THEN
			bControllerInRailDone:= TRUE;
			iStepAsm:= 120;			
		END_IF
		
	120:							//Wait until the rail is not in position
		IF NOT bRailReadyToAssembly OR bIn_ManualRun THEN
			iStepAsm:= 130;
		END_IF

	130:							//Return to start
		iStepAsm:= 0;

END_CASE
END_METHOD

METHOD PRIVATE Seq_CtrlCenter
VAR_INPUT
	bIsManual				: BOOL			:= FALSE;
END_VAR
CASE iStepCenter OF

	0:							//Reset variables		
		bCenterReadyToReceive:= FALSE;
		bCenterReadyToSend:= FALSE;
		tmrCenter.IN:= FALSE;
		iStepCenter:= 10;
				
	10:							//Check status
		IF bInSensorAfterFlipPos   THEN	//Controller in flipped/centering position
			//Avoid noise with the timer
			tmrCenter(IN:= TRUE, pt:= T#300MS);
			
			IF tmrCenter.Q THEN
				iStepCenter:= 40;
			END_IF				
					
		ELSE	//Nothing detected
			tmrCenter.IN:= FALSE;		
			iStepCenter:= 20;
		END_IF
	
	20:							//Confirm feed  cylinder retracted
		Cyl_FeedControl.bRetractRequest:= TRUE;
		IF Cyl_FeedControl.bIsRetracted THEN
			iStepCenter:= 30;
		END_IF
		
	30:							//Retract centering cylinder
		Cyl_Center.bRetractRequest:= TRUE;
		IF Cyl_Center.bIsRetracted THEN
			iStepCenter:= 40;
		END_IF
				
	40:							//Wait for controller in centering position 		
		bCenterReadyToReceive:= TRUE;
		IF bInSensorAfterFlipPos  THEN
			tmrAsm(IN:= TRUE, pt:= T#100MS);

			IF tmrAsm.Q THEN
				bCenterReadyToReceive:= FALSE;
				iStepCenter:= 50;
			END_IF						
		END_IF

	50:							//Confirm nothing to send
		IF NOT bReceiverReadyToSend THEN
			iStepCenter:= 60;
		END_IF

	60:							//Center controller
		 Cyl_Center.bExtendRequest:= TRUE;
		 IF Cyl_Center.bIsExtended THEN
			 	iStepCenter:= 70;
		 END_IF

	70:							//Centering cylinder retract
		Cyl_Center.bRetractRequest:= TRUE;
			IF Cyl_Center.bIsRetracted THEN
			 	iStepCenter:= 80;
		 	END_IF

	80:							//Wait for assembly to rail side ready to receive
		IF bAsmReadyToReceive THEN
			iStepCenter:= 90;
		END_IF
		
	90:							//Feed the controller to assembly side
		Cyl_FeedControl.bExtendRequest:= TRUE;
		IF Cyl_FeedControl.bIsExtended THEN
			//Update serial from the center position to the assembly
			sSerialAsm:= sSerialCenter;
			iStepCenter:= 100;
		END_IF
		
	100:						//Confirm controller in assembly position
		IF bInSensorAlignedPos THEN
			iStepCenter := 110;
		END_IF
		
	110:						//Retract feed cylinder
		Cyl_FeedControl.bRetractRequest:= TRUE;
		IF Cyl_FeedControl.bIsRetracted THEN
			iStepCenter:= 120;
		END_IF
			
	120:						//Wait for the ready to receive off
		bCenterReadyToSend:= FALSE;
		IF NOT bAsmReadyToReceive THEN
			iStepCenter:= 130;			
		END_IF

	130:						//Return to start
		iStepCenter:= 0;

END_CASE
END_METHOD

METHOD PRIVATE Seq_CtrlReceive
VAR_INPUT
	bIsManual				: BOOL		:= FALSE;
END_VAR

VAR
	
END_VAR
CASE iStepReceive OF

	0:							//Reset variables
		bOut_ReadyToRobotPlace:= FALSE;
		bReceiverReadyToSend:= FALSE;
		tmrFlip.IN:= FALSE;
		iStepReceive:= 10;
				
	10:							//Check status
	
		IF bInSensorBeforeFlipPos THEN	//Controller before flipped position
			//Avoid noise with the timer
			tmrFlip(IN:= TRUE, pt:= T#300MS);
			
			IF tmrFlip.Q THEN
				iStepReceive:= 40;
			END_IF				
		ELSIF bInSensorAfterFlipPos AND Vacuum.Vacuum_Ok THEN	//Controller in tool			
			//Avoid noise with the timer
			tmrFlip(IN:= TRUE, pt:= T#300MS);
			
			IF tmrFlip.Q THEN
				iStepReceive:= 60;
			END_IF
	
		ELSE	//Nothing detected		
			iStepReceive:= 20;
		END_IF
		
	20:							//Retract flipper to robot position	 
		
		Cyl_Flipper.bRetractRequest:= TRUE;
		IF Cyl_Flipper.bIsRetracted THEN
			iStepReceive:= 30;
		END_IF

	30:							//Send ready signal and wait for the new controller
		//Manual oper		 
		IF bIsManual THEN
			IF  bInSensorBeforeFlipPos THEN
				tmrFlip(IN:= TRUE, pt:= T#1S);
				IF tmrFlip.Q THEN	
					iStepReceive:= 40;
				END_IF
			ELSE
				tmrFlip(IN:= FALSE);
			END_IF
			
		//Automatic oper
		ELSE
			bOut_ReadyToRobotPlace:= TRUE;
			
			IF  bInSensorBeforeFlipPos THEN
				tmrFlip(IN:= TRUE, pt:= T#200MS);
				IF tmrFlip.Q THEN
					bOut_ReadyToRobotPlace:= FALSE;
					iStepReceive:= 40;	
				END_IF												
			END_IF							
		END_IF					
		
	40:		
		Vacuum.bGrip :=	TRUE;
		IF Vacuum.Vacuum_Ok THEN
			bReceiverReadyToSend:= TRUE;
			iStepReceive:= 50;
		END_IF

	50:							//Confirm centering side ready to receive						
		IF bCenterReadyToReceive THEN			
				iStepReceive := 60;			
		END_IF
				
	60:							//Flip controller	
		Cyl_Flipper.bExtendRequest:= TRUE;
		IF Cyl_Flipper.bIsExtended THEN
			iStepReceive := 70;
		END_IF
		
	70:							//Release controller	
		Vacuum.bGrip := FALSE; 							
		IF NOT Vacuum.Vacuum_Ok THEN	//Not used blowOK bc can be missed?
			//Update serial
			bReceiverReadyToSend:= FALSE;
			sSerialCenter:= sSerialReceived;		
			iStepReceive := 80;			
		END_IF
		
	80:							//Confirm controller in center side
		IF NOT bCenterReadyToReceive THEN
			iStepReceive:= 90;
		END_IF
						
	90:							//Return to start	
		iStepReceive := 0;
				
END_CASE
END_METHOD

METHOD Stop
fn_CancelCylinderMoves();
END_METHOD

METHOD UnclampRail : BOOL
VAR_INPUT
END_VAR
//Retract busbar support first
Cyl_BusbarSupport.bRetractRequest:= TRUE;
IF Cyl_BusbarSupport.bIsRetracted THEN
		
	//Top and bottom unclamp
	Cyl_ClampRail_Top.bRetractRequest:= TRUE;
	Cyl_ClampRail_Bot.bRetractRequest:= TRUE;
	IF Cyl_ClampRail_Top.bIsRetracted AND Cyl_ClampRail_Bot.bIsRetracted THEN	

		UnclampRail:= TRUE;		
		RETURN;			
	END_IF
END_IF
END_METHOD

END_FUNCTION_BLOCK

// ---- POUs/01-FunctionBlocks/MaterialSupply/FB_LoadStation.TcPOU
FUNCTION_BLOCK FB_LoadStation EXTENDS RACBaseObjects.FB_Machine
VAR_INPUT
	bDisableScan						: BOOL;
	bIn_MovePermisive					: BOOL;
	bIn_CvyStepDone						: BOOL;
	
	
END_VAR
VAR_OUTPUT
	bOut_ProcessDone						:BOOL;
END_VAR
VAR
	
	b_SensorLoadPos				AT %I*		: BOOL;	

	k50_Left								: RACBaseObjects.FB_Bimanual;
	k50_Right								: RACBaseObjects.FB_Bimanual;
	ScanerReinsertionLoad					: FB_Scanner;
	bSafeCurtainsFree			AT %I*		: BOOL;
	tmrCurtainsFree							: TON;
	b_SensorEndcap				AT %I* 		: BOOL;
	b_SensorController			AT %I*		: BOOL;
	
	b_IG_Sensor_Pass				AT %I*		: BOOL;
	b_IG_Sensor_Fail				AT %I*		: BOOL;
	Mtr_CenterLeft							: FB_Motor;
	Mtr_CenterRight							: FB_Motor;
	
	bScanController							: BOOL;
	bScanComplete							: BOOL;
	
	lr_WithEndcapPos							: LREAL;
	lr_WithoutEndcapPos						: LREAL;
	
	lr_WithControllerPos						: LREAL;
	lr_WithoutControllerPos					: LREAL;
	
	//Manual control
	b_MoveLeftMotor							: BOOL;
	b_MoveRightMotor						: BOOL;
	bIn_RailReady							: BOOL;
	
	
END_VAR

//Run the main control directly from the machine base
SUPER^.MachineMain();

{warning 'Add method implementation '}
METHOD Alarm
END_METHOD

{warning 'Add method implementation '}
METHOD Auto
IF diActualSeqStep<1000 OR diActualSeqStep> 2000 THEN
	diActualSeqStep:= 1000;
END_IF


CASE diActualSeqStep OF
	1000:						//Reset variables
		bScanController:= FALSE;
		bScanComplete:= FALSE;
		bOut_ProcessDone:= FALSE;
		
		Mtr_CenterLeft.bExecute:= FALSE;
		Mtr_CenterRight.bExecute:= FALSE;
		
		diActualSeqStep:= 1010;
	
		
	1010:						//Check status
		diActualSeqStep:= 1020;
		
	1020:						//Confirm motors not moving
		IF NOT Mtr_CenterLeft.bMotorMoving AND NOT Mtr_CenterRight.bMotorMoving THEN
			diActualSeqStep:= 1030;
		END_IF
		
	1030:						//Update motor params
		Mtr_CenterLeft.MovementType:= EN_MotionType.absolute;
		Mtr_CenterRight.MovementType:= EN_MotionType.absolute;
		
		Mtr_CenterLeft.lrPosition:= 0;
		Mtr_CenterRight.lrPosition:= 0;
		
		diActualSeqStep:= 1040;
		
	1040:						//Retract motors
		Mtr_CenterLeft.bExecute:= TRUE;
		Mtr_CenterRight.bExecute:= TRUE;
		
		IF Mtr_CenterLeft.bDone AND Mtr_CenterRight.bDone THEN
			Mtr_CenterLeft.bExecute := FALSE;
			Mtr_CenterRight.bExecute:= FALSE;
			diActualSeqStep:= 1050;
		END_IF	
	
	1050:						//Wait for the conveyor step
		IF bIn_CvyStepDone THEN
			diActualSeqStep:= 1060;
		END_IF
		
	1060:						//Check for the rail loaded
		IF b_SensorLoadPos AND bSafeCurtainsFree THEN
			diActualSeqStep:= 1070;
		END_IF
		
	1070:						//Validate banana effect/ IG sensor
	
		//Que haremos, esperar que se retire y se cargue otra?
		IF b_IG_Sensor_Pass THEN
			diActualSeqStep:= 1090;
		ELSIF b_IG_Sensor_Fail THEN
			diActualSeqStep:= 1080;
			sAlarm:= 'RailBanana, remove';
		END_IF
		
	1080:						//Rail on fail, wait until remove to return  to new load
		IF NOT b_SensorLoadPos THEN			
			diActualSeqStep:=1060;
		END_IF
	
	1090:						//Check reinsertion conditions
	
		Mtr_CenterLeft.MovementType:= EN_MotionType.absolute;
		Mtr_CenterRight.MovementType:= EN_MotionType.absolute;
		IF b_SensorEndcap THEN
			GVL_Rails.Nests[Constants.LoadPos].endcapAssembled := TRUE;
			Mtr_CenterRight.lrPosition:= lr_WithEndcapPos;
		ELSE
			Mtr_CenterRight.lrPosition:= lr_WithoutEndcapPos;
		END_IF
		
		IF b_SensorController THEN
			
			GVL_Rails.Nests[Constants.LoadPos].controllerAssembled := TRUE;
			//Start scanning on the IO task
			bScanController:= TRUE;
			Mtr_CenterLeft.lrPosition:= lr_WithControllerPos;
			
		ELSE
			Mtr_CenterLeft.lrPosition:= lr_WithoutControllerPos;
		END_IF
		
		diActualSeqStep:= 1100;

	1100:						//Move motors to center pos
		Mtr_CenterLeft.bExecute:= TRUE;
		Mtr_CenterRight.bExecute:= TRUE;

		IF Mtr_CenterLeft.bDone AND Mtr_CenterRight.bDone THEN			
			diActualSeqStep:= 1110;
		END_IF		
	
	1110:						//Confirm motors done false
		Mtr_CenterLeft.bExecute:= FALSE;
		Mtr_CenterRight.bExecute:= FALSE;
		IF NOT Mtr_CenterLeft.bDone AND NOT Mtr_CenterRight.bDone THEN
			diActualSeqStep:= 1120;
		END_IF
		
	1120:						//Wait 50 milis to confirm align
		Mtr_CenterLeft.lrPosition:= 0;
		Mtr_CenterRight.lrPosition:= 0;
		ton_StepTimeout(IN:= TRUE, PT:= T#50MS);
		
		IF ton_StepTimeout.Q THEN
			diActualSeqStep:= 1130;
		END_IF
		
	1130:						//Move motors to retract position	
	
		Mtr_CenterLeft.bExecute:= TRUE;
		Mtr_CenterRight.bExecute:= TRUE;
		
		IF Mtr_CenterLeft.bDone AND Mtr_CenterRight.bDone THEN
			diActualSeqStep:= 1140;
		END_IF
		
	1140:						//Check if there is a controller, wait for the scanned code
		IF b_SensorController  THEN
			IF bScanComplete THEN
				IF ScanerReinsertionLoad.sCode <> 'ERROR' THEN
					diActualSeqStep:= 1150;
				ELSE
					sAlarm:= 'Cant read the controller code, replace rail';
					
					diActualSeqStep:= 1080;		//Remove rail					
				END_IF
			END_IF
		ELSE
			diActualSeqStep:= 1150;			
		END_IF
		
	1150:						//Set the process done and wait for not rail ready
		bOut_ProcessDone:= TRUE;
		IF NOT bIn_RailReady THEN
			bOut_ProcessDone:= FALSE;
			diActualSeqStep:= 1160;
		END_IF
	
	1160:						//Return sequence
		diActualSeqStep:= 1000;
	

END_CASE
END_METHOD

METHOD fn_ReinsertionScanController : BOOL
VAR_INPUT
END_VAR
//Scanner disabled
IF ScanerReinsertionLoad.bDisable THEN
	GVL_Rails.Nests[Constants.LoadPos].controllerSerial:= 'ScanDisabled';
	GVL_Rails.Nests[Constants.LoadPos].okToProcess:= TRUE;
	fn_ReinsertionScanController:= TRUE;
	RETURN;
END_IF

//Get code
ScanerReinsertionLoad.bIn_Trigger:= TRUE;
IF ScanerReinsertionLoad.bCompleted  THEN
	ScanerReinsertionLoad.bIn_Trigger:= FALSE;
	
	GVL_Rails.Nests[Constants.LoadPos].controllerSerial:=ScanerReinsertionLoad.sCode;
	
	//If scan fails
	IF ScanerReinsertionLoad.sCode = 'ERROR' THEN
		GVL_Rails.Nests[Constants.LoadPos].okToProcess:= FALSE;
	END_IF
	
	fn_ReinsertionScanController:= TRUE;
END_IF
END_METHOD

{warning 'Add method implementation '}
METHOD Init
//Run timer for the timeouts
ton_StepTimeout();

CASE  diActualSeqStep OF
	0:						//Reset variables
		diActualSeqStep:= 10;
		
	10:						//Wait for initial move permisive
		IF Mtr_CenterLeft.bInit_StartPermissive AND Mtr_CenterRight.bInit_StartPermissive THEN
			diActualSeqStep:= 20;
		END_IF
		
	20:						//Check for the initial done reset
		IF NOT Mtr_CenterLeft.bInit_Finished AND NOT Mtr_CenterRight.bInit_Finished THEN
			diActualSeqStep:= 30;
		END_IF
		
		
	30:						//Motors home
		Mtr_CenterLeft.Init();
		Mtr_CenterRight.Init();
		ton_StepTimeout.IN:= TRUE;		
		//Wait for the initial finish
		IF Mtr_CenterLeft.bInit_Finished  AND Mtr_CenterRight.bInit_Finished THEN
			sAlarm:= '';
			ton_StepTimeout.IN:= FALSE;
			diActualSeqStep:= 40;
		
		//If timeoutm send the alarm
		ELSIF ton_StepTimeout.Q THEN
			IF NOT Mtr_CenterLeft.bInit_Finished THEN
				sAlarm:= 'Motor left didnt reach home position';
			ELSIF NOT Mtr_CenterRight.bInit_Finished THEN
				sAlarm:= 'Motor right didnt reach home position';
			END_IF
		END_IF
		
	40:						//Validate the scanner connection
		ton_StepTimeout.IN:= TRUE;
		IF ScanerReinsertionLoad.bConnected OR ScanerReinsertionLoad.bDisable THEN
			ton_StepTimeout.IN:= FALSE;
			diActualSeqStep:= 50;
		ELSIF ton_StepTimeout.Q THEN
			sAlarm:= 'Scanner not connected';
		END_IF
	
	50:						//Validate sensors
		//NOTE, validate for reset or how to confirm outputs
		diActualSeqStep:= 60;
		
	60:						//Spare
		diActualSeqStep:= 70;
		
	70:						//Send the initial finish
		bInit_Finished:= TRUE;
		
END_CASE
END_METHOD

{warning 'Add method implementation '}
METHOD IO
//Declare devices and add safety conditions
Mtr_CenterLeft(diStationState:= THIS^.diStationState,
				bInit_StartPermissive:= THIS^.bInit_StartPermissive and bSafeCurtainsFree,
				sDeviceID:= 'Mtr2',
				bStopExecution:= THIS^.bStopExecution,
				bAlarmReset:= THIS^.bAlarmReset,
				bMovePermissive:= THIS^.bIn_MovePermisive AND bSafeCurtainsFree);
				
Mtr_CenterRight(diStationState:= THIS^.diStationState,
				bInit_StartPermissive:= THIS^.bInit_StartPermissive AND bSafeCurtainsFree,
				sDeviceID:= 'Mtr2',
				bStopExecution:= THIS^.bStopExecution,
				bAlarmReset:= THIS^.bAlarmReset,
				bMovePermissive:= THIS^.bIn_MovePermisive AND bSafeCurtainsFree);
				
				

ScanerReinsertionLoad(bDisable:= bDisableScan, bAlarmReset:= bAlarmReset);

IF bScanController THEN
	IF THIS^.fn_ReinsertionScanController() THEN
		bScanController:=FALSE;
		bScanComplete:= TRUE;
	END_IF	

END_IF
END_METHOD

{warning 'Add method implementation '}
METHOD Manual
//Move motor left
IF b_MoveLeftMotor THEN
	Mtr_CenterLeft.bExecute:= TRUE;
	
	IF Mtr_CenterLeft.bDone THEN
		Mtr_CenterLeft.bExecute:= FALSE;
		b_MoveLeftMotor:= FALSE;
	END_IF
ELSE
	Mtr_CenterLeft.bExecute:= FALSE;	
END_IF

//Move motor right
IF b_MoveRightMotor THEN
	Mtr_CenterRight.bExecute:= TRUE;
	
	IF Mtr_CenterRight.bDone THEN
		Mtr_CenterRight.bExecute:= FALSE;
		b_MoveRightMotor:= FALSE;
	END_IF
ELSE
	Mtr_CenterRight.bExecute:= FALSE;	
END_IF
END_METHOD

{warning 'Add method implementation '}
METHOD Pause
END_METHOD

{warning 'Add method implementation '}
METHOD Stop
END_METHOD

END_FUNCTION_BLOCK
